KUKA KRL data list: RoboSyncStepper.dat

&ACCESS RVO3
&REL 16
&PARAM DISKPATH = KRC:\R1\TP\CNCRobotics\CEAD
DEFDAT  RoboSyncStepper PUBLIC
;************************************************
;     NextState Automation Ltd
;     www.nextstateautomation.co.uk
;************************************************
;     Contact: helpdesk@nextstate.co.uk
;     Date: 14/09/26
;     Version: 0.1.1
;************************************************

GLOBAL CONST INT RESET_ALARM_CODE=186
GLOBAL CONST INT ENABLE_DRIVE=159
GLOBAL CONST INT DISABLE_DRIVE=158
GLOBAL CONST INT COMMENCE_JOGGING=150
GLOBAL CONST INT STOP_JOGGING=216
GLOBAL CONST INT MOVE_RELATIVE_DISTANCE=102
GLOBAL CONST INT MOVE_ABSOLUTE_DISTANCE=103
GLOBAL CONST INT FAST_STOP_MOVE=225
GLOBAL CONST INT STOP_MOVE=226
GLOBAL CONST INT SET_POSITION = 165

GLOBAL ENUM ENUM_STEPPER_PARAM CURRENT,IDLE_CURRENT,PULSE_PER_REV,JOG_SPEED,JOG_ACCEL,JOG_DECEL,SPEED,ACCEL,DECEL,DISTANCE,SET_POSITION

ENDDAT
